// SIMATIC S7-200 SMART project (STEP 7-Micro/WIN SMART), CPU ST20

SYMBOL_TABLE 系统符号
Always_On        SM0.0    // 始终接通
END_SYMBOL_TABLE

ORGANIZATION_BLOCK MAIN:OB1
TITLE=程序注释
BEGIN
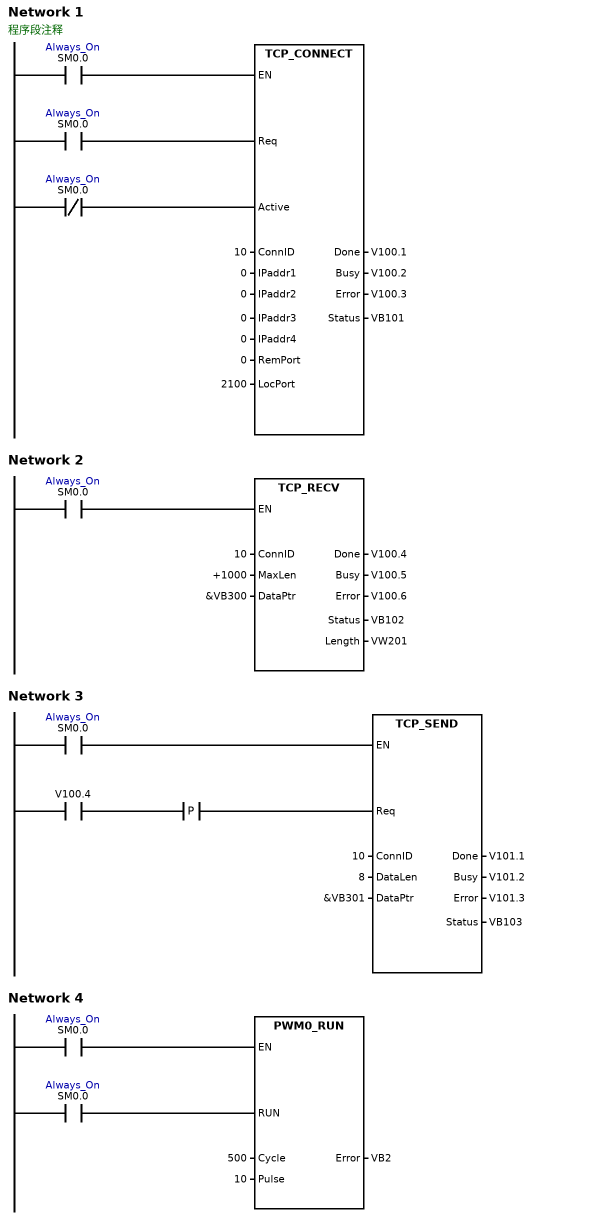
Network 1
// 程序段注释
LD     Always_On:SM0.0
=      L60.0
LD     Always_On:SM0.0
=      L63.7
LDN    Always_On:SM0.0
=      L63.6
LD     L60.0
CALL   TCP_CONNECT:SBR1, L63.7, L63.6, 10, 0, 0, 0, 0, 0, 2100, V100.1, V100.2, V100.3, VB101
Network 2
LD     Always_On:SM0.0
CALL   TCP_RECV:SBR2, 10, +1000, &VB300, V100.4, V100.5, V100.6, VB102, VW201
Network 3
// (network saved uncompiled; LAD cells follow)
// row 0: c0 -| |- Always_On:SM0.0  c1 --  c2 --  c3 [TCP_SEND EN:=power@row0, Req:=power@row1, ConnID:=10, DataLen:=8, DataPtr:=&VB301, Done=>V101.1, Busy=>V101.2, Error=>V101.3, Status=>VB103]
// row 1: c0 -| |- V100.4  c1 -|P|-  c2 --  c3 [box]
// row 2: c3 [box]
// row 3: c3 [box]
Network 4
LD     Always_On:SM0.0
=      L60.0
LD     Always_On:SM0.0
=      L63.7
LD     L60.0
CALL   PWM0_RUN:SBR3, L63.7, 500, 10, VB2
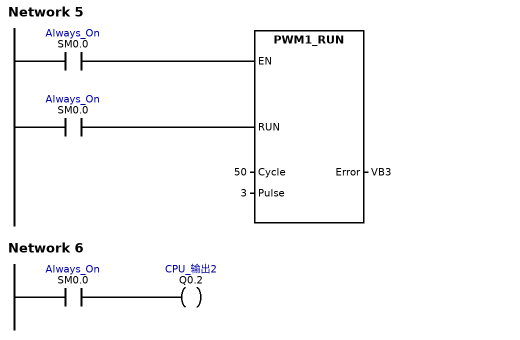
Network 5
LD     Always_On:SM0.0
=      L60.0
LD     Always_On:SM0.0
=      L63.7
LD     L60.0
CALL   PWM1_RUN:SBR4, L63.7, 50, 3, VB3
Network 6
LD     Always_On:SM0.0
=      CPU_输出2:Q0.2
END_ORGANIZATION_BLOCK

// SBR1: protected block, not included

// SBR2: protected block, not included

// SBR3: protected block, not included

// SBR4: protected block, not included

// SBR5: protected block, not included
